FUNCTION_BLOCK ReceptionRoom EXTENDS BaseRoom
VAR_INPUT
	rTemperature	: LREAL := 20.0 + Math.Random();
END_VAR
VAR    
    // Entity
    _entityExtend	: EntityExtend(_entityStart);
	
    _lowTemperature	: Room_State_LowTemperature(_ctx, rTemperature);
	
    _entityEnd2		: EntityEnd;
END_VAR

METHOD Execute
SUPER^.Execute();

// Simulation
IF NOT sim.bTick THEN
	RETURN;
END_IF

IF bInletValve AND bOutletValve THEN
	rTemperature := rTemperature + sim.param.rRoomTemperatureRisePerHeater * Math.Random();
END_IF

rTemperature := rTemperature + sim.param.rRoomTemperaturePassiveDrop * Math.Random();

IF rTemperature < 0 THEN
	rTemperature := 0;
ELSIF rTemperature > 100 THEN
	rTemperature := 100;
END_IF
END_METHOD

END_FUNCTION_BLOCK

(* stored: Version 1.1.0.1
   POU ReceptionRoom: Id {da0c2305-b67f-4452-8260-f7daed97569d}, SpecialFunc None
   Method Execute: Id {cebc7a85-aeea-43df-bbe1-0c63df1252f3} *)
